Xinje XCPPro project, PLC1: XC3-24 (software 3.3L)

PROGRAM Ladder

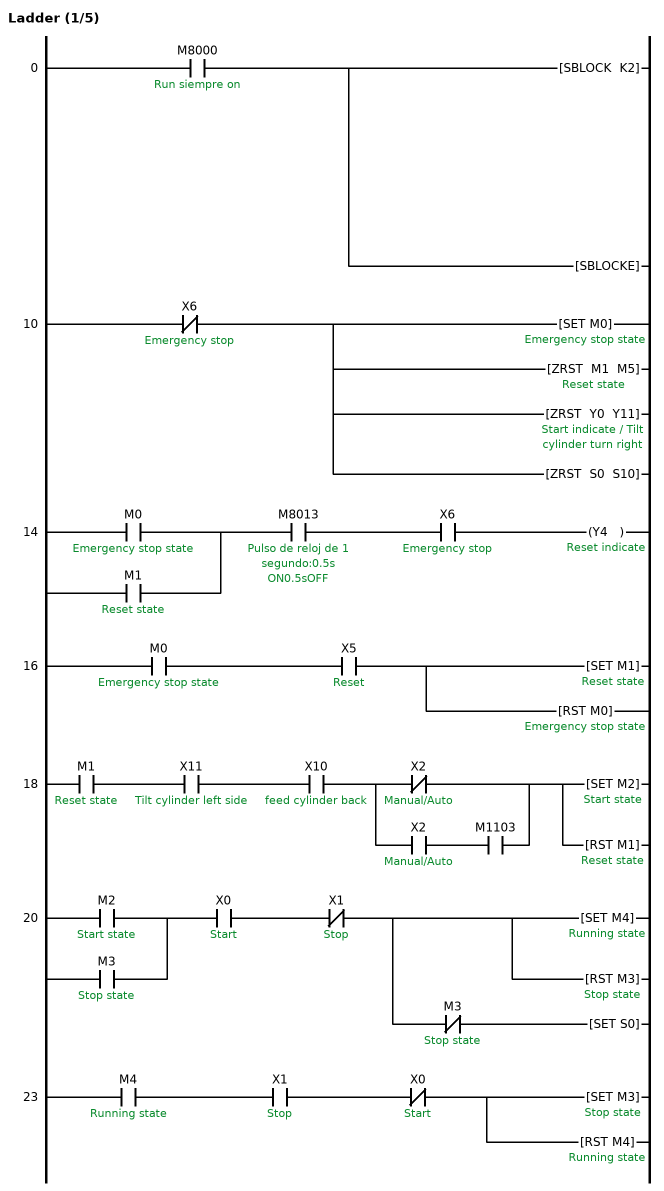
LD     M8000	; Run siempre on
SBLOCK K2
SBLOCKE
LDI    X6	; Emergency stop
SET    M0	; Emergency stop state
ZRST   M1 M5	; Reset state
ZRST   Y0 Y11	; Start indicate / Tilt cylinder turn right
ZRST   S0 S10
LD     M0	; Emergency stop state
OR     M1	; Reset state
AND    M8013	; Pulso de reloj de 1 segundo:0.5s ON0.5sOFF
AND    X6	; Emergency stop
OUT    Y4	; Reset indicate 
LD     M0	; Emergency stop state
AND    X5	; Reset
SET    M1	; Reset state
RST    M0	; Emergency stop state
LD     M1	; Reset state
AND    X11	; Tilt cylinder left side
AND    X10	; feed cylinder back
LDI    X2	; Manual/Auto
LD     X2	; Manual/Auto
AND    M1103
ORB
ANB
SET    M2	; Start state
RST    M1	; Reset state
LD     M2	; Start state
OR     M3	; Stop state
AND    X0	; Start
ANI    X1	; Stop
SET    M4	; Running state
RST    M3	; Stop state
ANI    M3	; Stop state
SET    S0
LD     M4	; Running state
AND    X1	; Stop
ANI    X0	; Start
SET    M3	; Stop state
RST    M4	; Running state

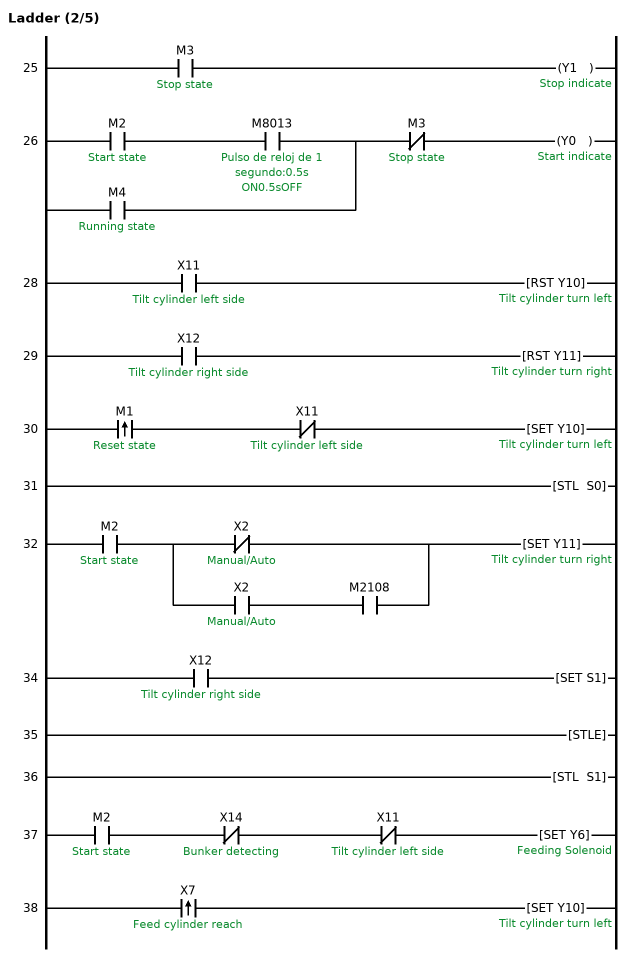
LD     M3	; Stop state
OUT    Y1	; Stop indicate
LD     M2	; Start state
AND    M8013	; Pulso de reloj de 1 segundo:0.5s ON0.5sOFF
OR     M4	; Running state
ANI    M3	; Stop state
OUT    Y0	; Start indicate
LD     X11	; Tilt cylinder left side
RST    Y10	; Tilt cylinder turn left
LD     X12	; Tilt cylinder right side
RST    Y11	; Tilt cylinder turn right
LDP    M1	; Reset state
ANI    X11	; Tilt cylinder left side
SET    Y10	; Tilt cylinder turn left
STL    S0
LD     M2	; Start state
LDI    X2	; Manual/Auto
LD     X2	; Manual/Auto
AND    M2108
ORB
ANB
SET    Y11	; Tilt cylinder turn right
LD     X12	; Tilt cylinder right side
SET    S1
STLE
STL    S1
LD     M2	; Start state
ANI    X14	; Bunker detecting
ANI    X11	; Tilt cylinder left side
SET    Y6	; Feeding Solenoid
LDP    X7	; Feed cylinder reach
SET    Y10	; Tilt cylinder turn left

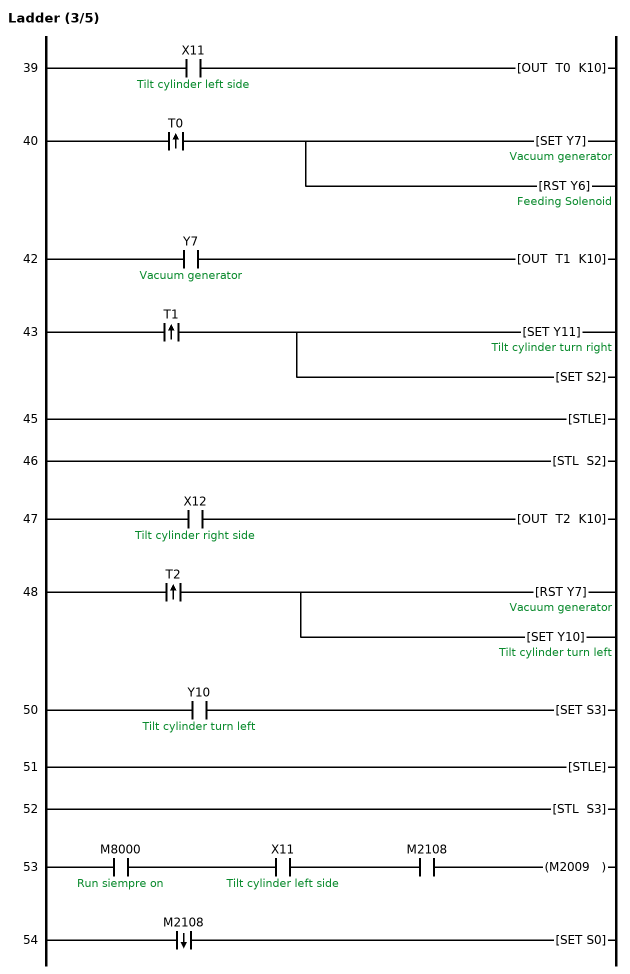
LD     X11	; Tilt cylinder left side
OUT    T0 K10
LDP    T0
SET    Y7	; Vacuum generator
RST    Y6	; Feeding Solenoid
LD     Y7	; Vacuum generator
OUT    T1 K10
LDP    T1
SET    Y11	; Tilt cylinder turn right
SET    S2
STLE
STL    S2
LD     X12	; Tilt cylinder right side
OUT    T2 K10
LDP    T2
RST    Y7	; Vacuum generator
SET    Y10	; Tilt cylinder turn left
LD     Y10	; Tilt cylinder turn left
SET    S3
STLE
STL    S3
LD     M8000	; Run siempre on
AND    X11	; Tilt cylinder left side
AND    M2108
OUT    M2009
LDF    M2108
SET    S0

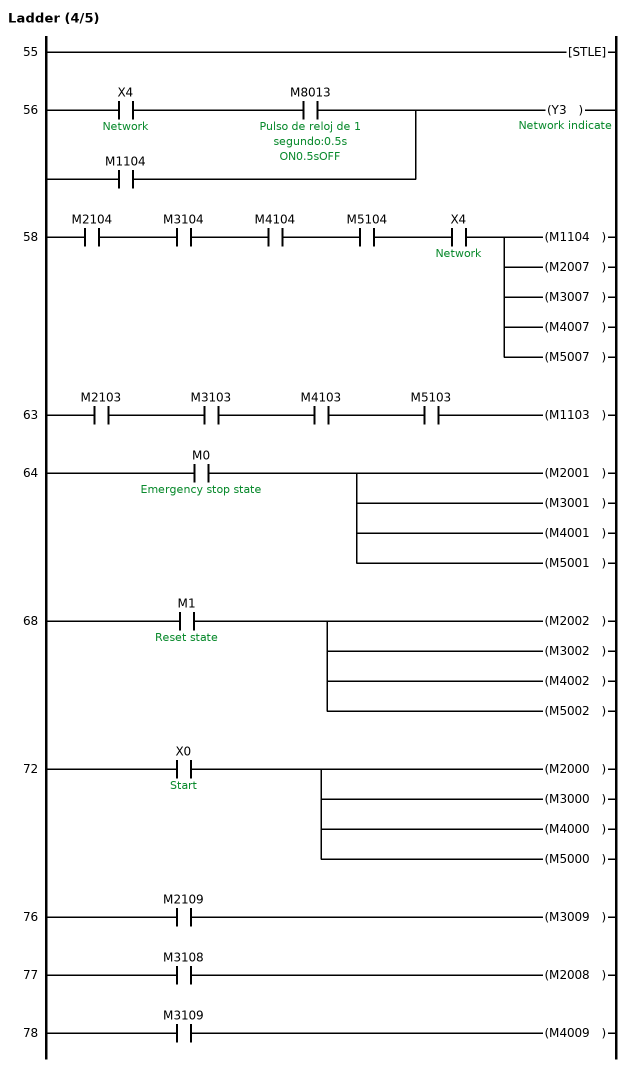
STLE
LD     X4	; Network
AND    M8013	; Pulso de reloj de 1 segundo:0.5s ON0.5sOFF
OR     M1104
OUT    Y3	; Network indicate
LD     M2104
AND    M3104
AND    M4104
AND    M5104
AND    X4	; Network
OUT    M1104
OUT    M2007
OUT    M3007
OUT    M4007
OUT    M5007
LD     M2103
AND    M3103
AND    M4103
AND    M5103
OUT    M1103
LD     M0	; Emergency stop state
OUT    M2001
OUT    M3001
OUT    M4001
OUT    M5001
LD     M1	; Reset state
OUT    M2002
OUT    M3002
OUT    M4002
OUT    M5002
LD     X0	; Start
OUT    M2000
OUT    M3000
OUT    M4000
OUT    M5000
LD     M2109
OUT    M3009
LD     M3108
OUT    M2008
LD     M3109
OUT    M4009

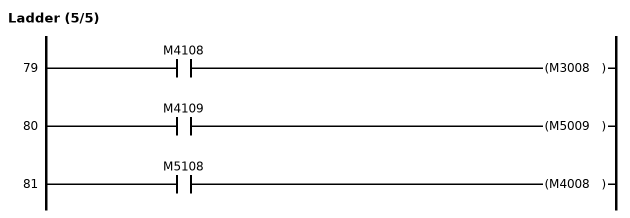
LD     M4108
OUT    M3008
LD     M4109
OUT    M5009
LD     M5108
OUT    M4008

COMMENTS (devices not used above)
X13	Vacuum pressure reach
Y5	Alarma de luz

SBLOCK K2	; 通信
  ; 2#检测写
  MCLW K2 K2000 K16 M2000 K2
  ; 3#装配写
  MCLW K3 K3000 K16 M3000 K2
  ; 4#冲压写
  MCLW K4 K4000 K16 M4000 K2
  ; 5#分拣写
  MCLW K5 K5000 K16 M5000 K2
  ; 2#检测读
  COLR K2 K2100 K16 M2100 K2
  ; 3#装配读
  COLR K3 K3100 K16 M3100 K2
  ; 4#冲压读
  COLR K4 K4100 K16 M4100 K2
  ; 5#分拣读
  COLR K5 K5100 K16 M5100 K2